{attribute 'GeneratedUsingTerminal: EL9221-4030-0018'}
{attribute addProperty BoxType "EL9221-4030-0018"}
{attribute addProperty Id "StatusAT %I*Status_FCAFFB9E11"}
{attribute addProperty CRC "2362336763"}
{attribute addProperty Size "11"}
TYPE OCP_Inputs_8CCE65FB EXTENDS InputBase_8311D824 :
STRUCT
	{attribute addProperty Name "Status"}
	Status AT %I* : Status_FCAFFB9E;
END_STRUCT
END_TYPE

(* stored: Version 1.2.0.0, ProductVersion 3.1.4024.11
   DUT OCP_Inputs_8CCE65FB: Id {f17084e5-a8dc-4aa1-82ac-05b66f83b1c8} *)
